// TIA Portal project "Automated_Sorting_Conveyor" (V17)

(* hardware
DEVICE "S7-1200 station_1"  S7-1200 Station
   slot 0: "Rack_0"  S7-1200 Rack  Rack  V1.0
   slot 1: "sort_conveyor"  CPU 1214C DC/DC/DC  6ES7 214-1AG40-0XB0  V4.5
   slot 2: "AQ 2x14BIT_1"  SM 1232 AQ2  6ES7 232-4HB32-0XB0  V2.1
DEVICE "HMI_1"  KTP700 Basic PN
   slot 0: "HMI_1"  KTP700 Basic PN  6AV2 123-2GB03-0AX0  17.0.0.0
   slot 1: "HMI_RT_1"  KTP700 Basic PN  6AV2 123-2GB03-0AX0  17.0.0.0
   slot 5: "HMI_1.IE_CP_1"  PROFINET Interface  17.0.0.0
      slot 1: "PROFINET Interface_1"  PROFINET Interface
         slot 1: "Port_1"  Port
DEVICE "SINAMICS G_1"  Sinamics.Device
   slot 0: "	_0"  Rail  SinamicsG120RackPN
   slot 0: "Drive_1"  G120 CU240E-2 PN  6SL3244-0BB12-1FA0  4.7.14
      slot 1: "PROFINET interface"  MDD-SinamicsG120-P
   slot 3: "PM240 IP20"  PM240 IP20  6SL3224-0BE13-7UA0  -
*)

// ===== PLC "sort_conveyor"  CPU 1214C DC/DC/DC =====

VAR_GLOBAL   // PLC tag table "PLC_IO"
   "PB_Start" AT %I0.0 : Bool;   // Green push button (NO)
   "PB_Stop" AT %I0.1 : Bool;   // Red push button (NC)
   "Safety_EStop" AT %I0.2 : Bool;   // Emergency Stop (NC)
   "Light_Curtain_OK" AT %I0.3 : Bool;   // Light curtain status (NC - TRUE when safe)
   "Sensor_Sort_Zone" AT %I0.4 : Bool;   // Detects box is in position
   "Sensor_Tall" AT %I0.5 : Bool;   // Photoelectric (Through-beam)
   "Sensor_Short" AT %I0.6 : Bool;   // Retro-reflective
   "Cyl_Pusher_Home" AT %I0.7 : Bool;   // Magnetic reed switch (Retracted)
   "Cyl_Pusher_Extended" AT %I1.0 : Bool;   // Magnetic reed switch (Extended)
   "VFD_Belt_A_Run" AT %Q0.0 : Bool;   // Command to VFD
   "VFD_Belt_B_Run" AT %Q0.1 : Bool;   // Command to VFD
   "Valve_Pusher_Extend" AT %Q0.2 : Bool;   // Solenoid valve
   "Alarm_Beacon_Red" AT %Q0.3 : Bool;   // Fault indication
   "Alarm_Beacon_Yellow" AT %Q0.4 : Bool;   // Warning/Running
   "VFD_Belt_A_Speed" AT %QW96 : Int;   // 0-10V speed reference (0-1000 RPM)
END_VAR

DATA_BLOCK "FB_Sorting_Conveyor_DB"   // DB2
{ S7_Optimized_Access := 'TRUE' }
VERSION : 0.1
// stored: InstanceOfName FB_Sorting_Conveyor
"FB_Sorting_Conveyor"
BEGIN
END_DATA_BLOCK

DATA_BLOCK "TO_Conveyor_Belt_A"   // DB1, Motion_DB
{ S7_Optimized_Access := 'TRUE' }
AUTHOR : SIMATIC
FAMILY : BasicMC
NAME : TO_PosAx
VERSION : 8.0
// stored: InstanceOfName TO_PositioningAxis
"TO_PositioningAxis"
BEGIN
   // Axis.EnableOutput_AddressCU = %Q0.0
   // Axis.AnalogOutput_AddressCU = %QW96
   // Axis.LengthUnitNormalized.Distance = 1013
   // Axis.Encoder.SelectedHscIndexCU = -1
   // Axis.Encoder.DbTypeCU = Classic
   // Axis.Drive.DbTypeCU = Classic
END_DATA_BLOCK

FUNCTION_BLOCK "FB_Sorting_Conveyor"   // FB1, SCL
{ S7_Optimized_Access := 'TRUE' }
VERSION : 0.1
   VAR
      Current_Step : Int;   // Grafcet step number
      Previous_Step : Int := -1;
      bAxisEnabled : Bool;   // MC_Power status
      bPowerBusy : Bool;   // MC_Power busy flag
      bPowerError : Bool;   // MC_Power error flag
      bMoveBusy : Bool;   // MC_MoveVelocity busy
      bMoveError : Bool;   // MC_MoveVelocity error
      bInVelocity : Bool;
      AxisPowerCmd : Bool;
      Fault_Active : Bool;   // System fault flag
      MoveCmd : Bool;
      ResetCmd : Bool;
      MoveVelocity : Real := 500.0;
      MoveDirection : Int := 1;
      LastErrorID : Word;
      LastErrorInfo : Word;
      Timer_Fault : TON_TIME;   // Fault detection timer
      MC_Power_FB : MC_Power;
      MC_MoveVel_FB : MC_MoveVelocity;
      MC_Reset_FB : MC_Reset;
      Reset_Pulse : Bool;
      xResetDone : Bool;
      Move_Execute_Pulse : Bool;
   END_VAR
BEGIN

   //========================================================
   // SAFETY
   //========================================================

   IF (NOT "Safety_EStop") OR (NOT "Light_Curtain_OK") THEN

       #Fault_Active := TRUE;

       #AxisPowerCmd := FALSE;
       #MoveCmd := FALSE;
       #ResetCmd := FALSE;   // don't force reset while the fault is still present

       "Valve_Pusher_Extend" := FALSE;
       "VFD_Belt_B_Run" := FALSE;
       "VFD_Belt_A_Run" := FALSE;
       "VFD_Belt_A_Speed" := 0;

       "Alarm_Beacon_Red" := TRUE;
       "Alarm_Beacon_Yellow" := FALSE;

       // Route straight to the fault/stopped state instead of an undefined step.
       #Current_Step := 99;

   END_IF;

   //========================================================
   // STEP CHANGE DETECTION
   //========================================================

   IF #Current_Step <> #Previous_Step THEN

       #MoveCmd := FALSE;
       #ResetCmd := FALSE;
       #Reset_Pulse := FALSE;

   END_IF;

   //=====================================================
   // GRAFCET
   //=====================================================

   CASE #Current_Step OF

           //-----------------------------------------------------
           // STEP 0 - Idle
           //-----------------------------------------------------
       0:

           #MC_Power_FB(
                        Axis := "TO_Conveyor_Belt_A",
                        Enable := FALSE,
                        StartMode := 1,
                        StopMode := 0,
                        Status => #bAxisEnabled,
                        Busy => #bPowerBusy,
                        Error => #bPowerError);

           "Valve_Pusher_Extend" := FALSE;
           "VFD_Belt_B_Run" := FALSE;
           "VFD_Belt_A_Run" := FALSE;
           "VFD_Belt_A_Speed" := 0;

           "Alarm_Beacon_Red" := FALSE;
           "Alarm_Beacon_Yellow" := FALSE;

           #Fault_Active := FALSE;
           #bInVelocity := FALSE;

           // Clear any latent axis error left over from a fault before allowing a start.
           IF #MC_Power_FB.Error THEN

               #MC_Reset_FB(
                            Axis := "TO_Conveyor_Belt_A",
                            Execute := TRUE,
                            Done => #xResetDone);

           ELSE

               #MC_Reset_FB(
                            Axis := "TO_Conveyor_Belt_A",
                            Execute := FALSE);

           END_IF;

           IF "PB_Start" AND "Cyl_Pusher_Home" AND (NOT #MC_Power_FB.Error) THEN
               #Current_Step := 10;
           END_IF;



           //-----------------------------------------------------
           // STEP 10 - Belt A running, waiting for a part
           //-----------------------------------------------------

       10:

           // Generate rising edge for Move command (ONE SCAN ONLY)
           IF #Current_Step = 10 AND #Previous_Step <> 10 THEN
               #Move_Execute_Pulse := TRUE;
           ELSE
               #Move_Execute_Pulse := FALSE;
           END_IF;

           // Enable the axis
           #MC_Power_FB(
                        Axis := "TO_Conveyor_Belt_A",
                        Enable := TRUE,
                        StartMode := 1,
                        StopMode := 0,
                        Status => #bAxisEnabled,
                        Busy => #bPowerBusy,
                        Error => #bPowerError);

           // Move at velocity (with rising edge Execute)
           #MC_MoveVel_FB(
                          Axis := "TO_Conveyor_Belt_A",
                          Execute := #Move_Execute_Pulse,  // ← ONE SCAN ONLY!
                          Velocity := #MoveVelocity,
                          Direction := #MoveDirection,
                          Current := FALSE,
                          PositionControlled := TRUE,
                          Busy => #bMoveBusy,
                          Error => #bMoveError,
                          InVelocity => #bInVelocity);

           // Map to physical VFD outputs
           "VFD_Belt_A_Run" := #bAxisEnabled;
           "VFD_Belt_A_Speed" := REAL_TO_INT(#MoveVelocity);

           "Alarm_Beacon_Yellow" := TRUE;

           // Error handling
           IF #MC_Power_FB.Error OR #MC_MoveVel_FB.Error THEN
               #LastErrorID := #MC_MoveVel_FB.ErrorID;
               #LastErrorInfo := #MC_MoveVel_FB.ErrorInfo;
               #Current_Step := 99;
               // Transition to sorting when box detected
           ELSIF "Sensor_Sort_Zone" THEN
               #Current_Step := 20;
           END_IF;
           //-----------------------------------------------------
           // STEP 20 - Decelerate to stop, identify part height
           //-----------------------------------------------------
       20:

           #MC_MoveVel_FB(
                          Axis := "TO_Conveyor_Belt_A",
                          Execute := TRUE,
                          Velocity := 0.0,
                          Direction := #MoveDirection,
                          Current := FALSE,
                          PositionControlled := TRUE,
                          Busy => #bMoveBusy,
                          Error => #bMoveError,
                          InVelocity => #bInVelocity);

           "VFD_Belt_A_Run" := #bAxisEnabled;
           "VFD_Belt_A_Speed" := 0;

           #Timer_Fault(
                        IN := TRUE,
                        PT := T#3S);

           IF "Sensor_Tall" THEN

               #Timer_Fault(IN := FALSE,
                            PT := T#3S);
               #Current_Step := 30;

           ELSIF "Sensor_Short" THEN

               #Timer_Fault(IN := FALSE,
                            PT := T#3S);
               #Current_Step := 40;

           ELSIF #Timer_Fault.Q THEN

               #Timer_Fault(IN := FALSE,
                            PT := T#3S);
               #LastErrorID := 16#1001;   // custom: no part detected in time
               #Current_Step := 99;

           END_IF;


           //-----------------------------------------------------
           // STEP 30 - Tall part: pass straight through
           //-----------------------------------------------------
       30:

           // Generate rising edge for resume command
           IF #Current_Step = 30 AND #Previous_Step <> 30 THEN
               #Move_Execute_Pulse := TRUE;
           ELSE
               #Move_Execute_Pulse := FALSE;
           END_IF;

           #MC_MoveVel_FB(
                          Axis := "TO_Conveyor_Belt_A",
                          Execute := #Move_Execute_Pulse,  // ← ONE SCAN ONLY!
                          Velocity := #MoveVelocity,
                          Direction := #MoveDirection,
                          Current := FALSE,
                          PositionControlled := TRUE,
                          Busy => #bMoveBusy,
                          Error => #bMoveError,
                          InVelocity => #bInVelocity);

           "VFD_Belt_A_Run" := #bAxisEnabled;
           "VFD_Belt_A_Speed" := REAL_TO_INT(#MoveVelocity);

           // Wait for box to clear
           IF NOT "Sensor_Sort_Zone" THEN
               #Current_Step := 10;
           END_IF;

           //-----------------------------------------------------
           // STEP 40 - Short part: push off belt (extend)
           //-----------------------------------------------------
       40:

           "Valve_Pusher_Extend" := TRUE;

           IF "Cyl_Pusher_Extended" THEN
               #Current_Step := 41;
           END_IF;



           //-----------------------------------------------------
           // STEP 41 - Retract pusher
           //-----------------------------------------------------
       41:

           "Valve_Pusher_Extend" := FALSE;

           IF "Cyl_Pusher_Home" THEN
               #Current_Step := 42;
           END_IF;


           //-----------------------------------------------------
           // STEP 42 - Resume belt after push cycle
           //-----------------------------------------------------
       42:

           // Generate rising edge for resume command
           IF #Current_Step = 42 AND #Previous_Step <> 42 THEN
               #Move_Execute_Pulse := TRUE;
           ELSE
               #Move_Execute_Pulse := FALSE;
           END_IF;

           #MC_MoveVel_FB(
                          Axis := "TO_Conveyor_Belt_A",
                          Execute := #Move_Execute_Pulse,  // ← ONE SCAN ONLY!
                          Velocity := #MoveVelocity,
                          Direction := #MoveDirection,
                          Current := FALSE,
                          PositionControlled := TRUE,
                          Busy => #bMoveBusy,
                          Error => #bMoveError,
                          InVelocity => #bInVelocity);

           "VFD_Belt_A_Run" := #bAxisEnabled;
           "VFD_Belt_A_Speed" := REAL_TO_INT(#MoveVelocity);

           // Wait for box to clear
           IF NOT "Sensor_Sort_Zone" THEN
               #Current_Step := 10;
           END_IF;



           //-----------------------------------------------------
           // STEP 99 - Fault / Stopped
           //-----------------------------------------------------
       99:

           #MC_Power_FB(
                        Axis := "TO_Conveyor_Belt_A",
                        Enable := FALSE,
                        StartMode := 1,
                        StopMode := 0,
                        Status => #bAxisEnabled,
                        Busy => #bPowerBusy,
                        Error => #bPowerError);

           "Valve_Pusher_Extend" := FALSE;
           "VFD_Belt_B_Run" := FALSE;
           "VFD_Belt_A_Run" := FALSE;
           "VFD_Belt_A_Speed" := 0;

           "Alarm_Beacon_Red" := TRUE;
           "Alarm_Beacon_Yellow" := FALSE;

           #bInVelocity := FALSE;

           IF "PB_Stop"
               AND "Safety_EStop"
               AND "Light_Curtain_OK" THEN

               #Current_Step := 0;

           END_IF;

   END_CASE;

   #Previous_Step := #Current_Step;
END_FUNCTION_BLOCK

ORGANIZATION_BLOCK "Main"   // OB1, LAD, ProgramCycle
TITLE = "Main Program Sweep (Cycle)"
{ S7_Optimized_Access := 'TRUE' }
VERSION : 0.1
   VAR_INPUT
      Initial_Call : Bool;   // Initial call of this OB
      Remanence : Bool;   // =True, if remanent data are available
   END_VAR
BEGIN

REGION Network 1
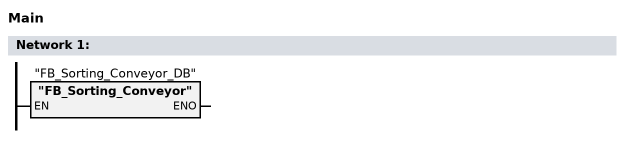
   RUNG wire#powerrail
      "FB_Sorting_Conveyor_DB"()
   END_RUNG
   // the same network as SCL:
   "FB_Sorting_Conveyor_DB"();   // "FB_Sorting_Conveyor"
END_REGION

REGION Network 2 (SCL): BELT B Control
   IF "Valve_Pusher_Extend" OR "Cyl_Pusher_Extended" THEN
       "VFD_Belt_B_Run" := TRUE;
   ELSE
       "VFD_Belt_B_Run" := FALSE;
   END_IF;
END_REGION
END_ORGANIZATION_BLOCK

(* ===== HMI "HMI_RT_1" =====
system functions are stored by id; their names below are inferred from use

HMI tags "Default tag table"
   "Tag_ScreenNumber" : UInt, internal

Template "Template_1" 800x480
   Button "Exit" at 714,429 size 71x50; TextOff 'Exit'; PictureOff "ExitRuntime_KTP700_Basic_PN_TR"; PictureOn "ExitRuntime_KTP700_Basic_PN_TR"
      on Release: StopRuntime(0)
   Button "Template_Button" at 614,429 size 71x50; TextOff 'Text'
   Button "Template_Button_1" at 514,429 size 71x50; TextOff 'Text'
   Button "Template_Button_2" at 414,429 size 71x50; TextOff 'Text'
   Button "Template_Button_3" at 314,429 size 71x50; TextOff 'Text'
   Button "Template_Button_4" at 214,429 size 71x50; TextOff 'Text'
   Button "Template_Button_5" at 114,429 size 71x50; TextOff 'Text'
   Button "Start screen" at 14,429 size 71x50; TextOff 'Start screen'; PictureOff "NavigateHome_KTP700_Basic_PN_TR"; PictureOn "NavigateHome_KTP700_Basic_PN_TR"
      on Release: ActivateScreen("Root screen", 0)
   SymbolicIOField "Symbolic_IO_Field_Screen" at 93,9 size 600x33; TextOff '0'; TextOn '1'; TextList "TextList_ScreenNames"
      ProcessValue <- "Tag_ScreenNumber"
      on Change: ActivateScreenByNumber("Tag_ScreenNumber", 0)
   DateTimeField "HmiScreenItemData" at 695,25 size 105x25
   DateTimeField "HmiScreenItemData_1" at 695,0 size 105x25
   GraphicView "Logo" at 0,0 size 91x51; Picture "Logo of HMI_1"

screen "Root screen" 800x480, template "Template_1"
   on GenerateScreen: SetTag("Tag_ScreenNumber", 1)
   TextField "HmiScreenItemData" at 80,225 size 640x25; Text 'Welcome to HMI_1 (KTP700 Basic+ PN)!'
*)